// LS Electric XG5000 project: Laser Film Ablation System
// PLC NewPLC

PROGRAM NewProgram (task: 스캔 프로그램)

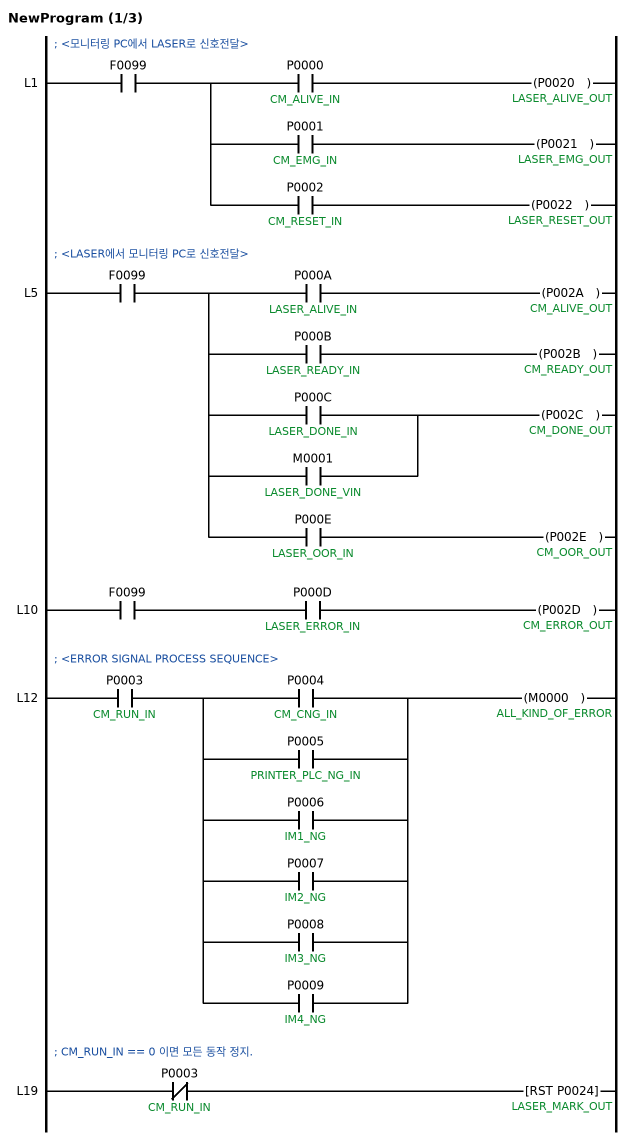
// <모니터링 PC에서 LASER로 신호전달>
; L1
LOAD      F0099
MPUSH
AND       P0000	// CM_ALIVE_IN
OUT       P0020	// LASER_ALIVE_OUT
MLOAD
AND       P0001	// CM_EMG_IN
OUT       P0021	// LASER_EMG_OUT
MPOP
AND       P0002	// CM_RESET_IN
OUT       P0022	// LASER_RESET_OUT
// <LASER에서 모니터링 PC로 신호전달>
; L5
LOAD      F0099
MPUSH
AND       P000A	// LASER_ALIVE_IN
OUT       P002A	// CM_ALIVE_OUT
MLOAD
AND       P000B	// LASER_READY_IN
OUT       P002B	// CM_READY_OUT
MLOAD
LOAD      P000C	// LASER_DONE_IN
OR        M0001	// LASER_DONE_VIN
AND LOAD
OUT       P002C	// CM_DONE_OUT
MPOP
AND       P000E	// LASER_OOR_IN
OUT       P002E	// CM_OOR_OUT
; L10
LOAD      F0099
AND       P000D	// LASER_ERROR_IN
OUT       P002D	// CM_ERROR_OUT
// <ERROR SIGNAL PROCESS SEQUENCE>
; L12
LOAD      P0003	// CM_RUN_IN
LOAD      P0004	// CM_CNG_IN
OR        P0005	// PRINTER_PLC_NG_IN
OR        P0006	// IM1_NG
OR        P0007	// IM2_NG
OR        P0008	// IM3_NG
OR        P0009	// IM4_NG
AND LOAD
OUT       M0000	// ALL_KIND_OF_ERROR
// CM_RUN_IN == 0 이면 모든 동작 정지.
; L19
LOAD NOT  P0003	// CM_RUN_IN
RST       P0024	// LASER_MARK_OUT

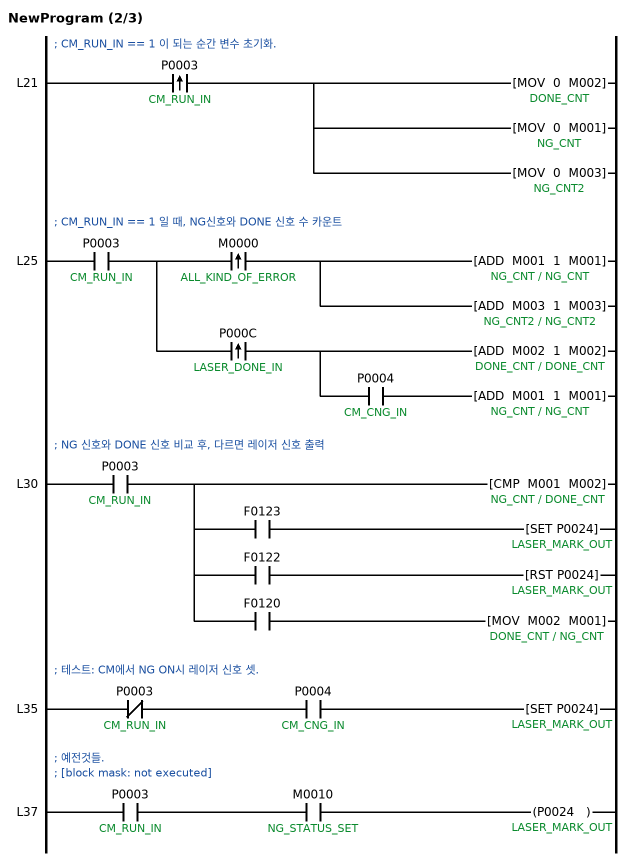
// CM_RUN_IN == 1 이 되는 순간 변수 초기화.
; L21
LOADP     P0003	// CM_RUN_IN
MOV       0 M002	// DONE_CNT
MOV       0 M001	// NG_CNT
MOV       0 M003	// NG_CNT2
// CM_RUN_IN == 1 일 때, NG신호와 DONE 신호 수 카운트
; L25
LOAD      P0003	// CM_RUN_IN
MPUSH
ANDP      M0000	// ALL_KIND_OF_ERROR
ADD       M001 1 M001	// NG_CNT / NG_CNT
ADD       M003 1 M003	// NG_CNT2 / NG_CNT2
MPOP
ANDP      P000C	// LASER_DONE_IN
ADD       M002 1 M002	// DONE_CNT / DONE_CNT
AND       P0004	// CM_CNG_IN
ADD       M001 1 M001	// NG_CNT / NG_CNT
// NG 신호와 DONE 신호 비교 후, 다르면 레이저 신호 출력
; L30
LOAD      P0003	// CM_RUN_IN
CMP       M001 M002	// NG_CNT / DONE_CNT
MPUSH
AND       F0123
SET       P0024	// LASER_MARK_OUT
MLOAD
AND       F0122
RST       P0024	// LASER_MARK_OUT
MPOP
AND       F0120
MOV       M002 M001	// DONE_CNT / NG_CNT
// 테스트: CM에서 NG ON시 레이저 신호 셋.
; L35
LOAD NOT  P0003	// CM_RUN_IN
AND       P0004	// CM_CNG_IN
SET       P0024	// LASER_MARK_OUT
// 예전것들.
; L37 (block mask: not executed)
LOAD      P0003	// CM_RUN_IN
AND       M0010	// NG_STATUS_SET
OUT       P0024	// LASER_MARK_OUT

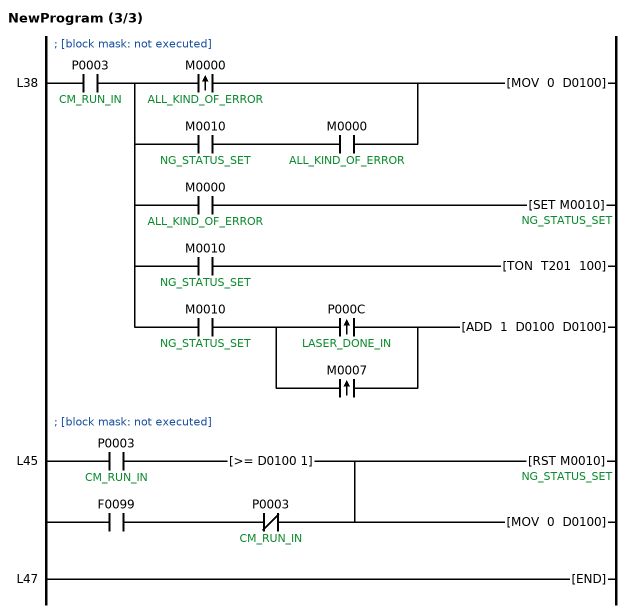
; L38 (block mask: not executed)
LOAD      P0003	// CM_RUN_IN
MPUSH
LOADP     M0000	// ALL_KIND_OF_ERROR
LOAD      M0010	// NG_STATUS_SET
AND       M0000	// ALL_KIND_OF_ERROR
OR LOAD
AND LOAD
MOV       0 D0100
MLOAD
AND       M0000	// ALL_KIND_OF_ERROR
SET       M0010	// NG_STATUS_SET
MLOAD
AND       M0010	// NG_STATUS_SET
TON       T201 100
MPOP
AND       M0010	// NG_STATUS_SET
LOADP     P000C	// LASER_DONE_IN
ORP       M0007
AND LOAD
ADD       1 D0100 D0100
; L45 (block mask: not executed)
LOAD      P0003	// CM_RUN_IN
AND>=     D0100 1
LOAD      F0099
AND NOT   P0003	// CM_RUN_IN
OR LOAD
RST       M0010	// NG_STATUS_SET
MOV       0 D0100
; L47
END

VARIABLES AND COMMENTS (devices not used above)
P0002F	BIT	CM_LOTCLEARDONE_OUT
P0000F	BIT	CM_LOTCLEAR_IN
P00025	BIT	LASER_LOTCLEAR_OUT
C0000	BIT/WORD	LASER_ON_COUNT